TYPE TcoAiStatus :
STRUCT
	{attribute addProperty Name "<#Raw range#>"}
	RawRange: REAL;
	{attribute addProperty Name "<#Real range#>"}
	RealRange: REAL;
	
	{attribute addProperty Name "<#Scaled value#>"}
	Scaled: REAL;
	
	
	
	
END_STRUCT
END_TYPE

(* stored: Version 1.1.0.1, ProductVersion 3.1.4024.9
   DUT TcoAiStatus: Id {4770b4bd-629a-0b04-102f-20faa737d5b4} *)
